FUNCTION_BLOCK OPCUA_VARIABLE_LIST_SAMPLING
  {SET_ATTRIBUTE(OpcUa, DEVICE.SENSOR)}
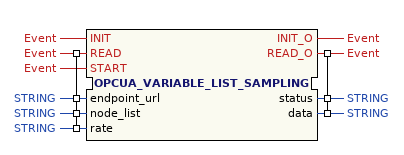
  EVENT_INPUT
    INIT;
    READ WITH endpoint_url, node_list, rate; {SET_ATTRIBUTE(OpcUa, Method)}
    START;
  END_EVENT
  EVENT_OUTPUT
    INIT_O;
    READ_O WITH status, data;
  END_EVENT
  VAR_INPUT
    endpoint_url : STRING; {SET_ATTRIBUTE(OpcUa, Constant)}
    node_list : STRING; {SET_ATTRIBUTE(OpcUa, Constant)}
    rate : STRING; {SET_ATTRIBUTE(OpcUa, Constant)}
  END_VAR
  VAR_OUTPUT
    status : STRING; {SET_ATTRIBUTE(OpcUa, Variable)}
    data : STRING; {SET_ATTRIBUTE(OpcUa, Variable)}
  END_VAR
END_FUNCTION_BLOCK
